// TIA Portal V20 export
TYPE "LER_typePartData"
// stored: Access Published
   STRUCT
      Common : "LER_typeCommonData";
      UnitData : "LER_typeUnitData";
   END_STRUCT;
END_TYPE
